LIN {X 0,Y 79.279,Z 952.165,A -85,B 0,C 180,E1 -27804.907,E2 -27804.907} C_VEL
LIN {X 0,Y 79.771,Z 953.591,A -85,B 0,C 180,E1 -27809.992,E2 -27809.992} C_VEL
LIN {X 0,Y 79.062,Z 954.279,A -85,B 0,C 180,E1 -27815.092,E2 -27815.092} C_VEL
LIN {X 0,Y 78.713,Z 954.565,A -85,B 0,C 180,E1 -27820.843,E2 -27820.843} C_VEL
LIN {X 0,Y 79.833,Z 953.994,A -85,B 0,C 180,E1 -27830.61,E2 -27830.61} C_VEL
LIN {X 0,Y 83.593,Z 951.93,A -85,B 0,C 180,E1 -27840.286,E2 -27840.286} C_VEL
LIN {X 0,Y 89.84,Z 948.411,A -85,B 0,C 180,E1 -27848.734,E2 -27848.734} C_VEL
LIN {X 0,Y 95.728,Z 944.699,A -85,B 0,C 180,E1 -27854.214,E2 -27854.214} C_VEL
LIN {X 0,Y 102.501,Z 939.995,A -85,B 0,C 180,E1 -27858.948,E2 -27858.948} C_VEL
LIN {X 0,Y 111.32,Z 933.115,A -85,B 0,C 180,E1 -27863.595,E2 -27863.595} C_VEL
LIN {X 0,Y 119.532,Z 925.735,A -85,B 0,C 180,E1 -27866.903,E2 -27866.903} C_VEL
LIN {X 0,Y 128.167,Z 916.709,A -85,B 0,C 180,E1 -27869.718,E2 -27869.718} C_VEL
LIN {X 0,Y 136.383,Z 906.598,A -85,B 0,C 180,E1 -27871.932,E2 -27871.932} C_VEL
LIN {X 0,Y 144.035,Z 895.124,A -85,B 0,C 180,E1 -27873.702,E2 -27873.702} C_VEL
LIN {X 0,Y 150.323,Z 883.666,A -85,B 0,C 180,E1 -27874.926,E2 -27874.926} C_VEL
LIN {X 0,Y 151.627,Z 880.908,A -85,B 0,C 180,E1 -27875.173,E2 -27875.173} C_VEL
LIN {X 0,Y 153.739,Z 875.695,A -85,B 0,C 180,E1 -27875.804,E2 -27875.804} C_VEL
LIN {X 0,Y 156.331,Z 867.052,A -85,B 0,C 180,E1 -27877.327,E2 -27877.327} C_VEL
LIN {X 0,Y 157.97,Z 860.05,A -85,B 0,C 180,E1 -27878.573,E2 -27878.573} C_VEL
LIN {X 0,Y 159.532,Z 852.692,A -85,B 0,C 180,E1 -27879.471,E2 -27879.471} C_VEL
LIN {X 0,Y 161.008,Z 844.469,A -85,B 0,C 180,E1 -27880.228,E2 -27880.228} C_VEL
LIN {X 0,Y 160.722,Z 839.975,A -85,B 0,C 180,E1 -27882.77,E2 -27882.77} C_VEL
LIN {X 0,Y 160.581,Z 836.729,A -85,B 0,C 180,E1 -27885.204,E2 -27885.204} C_VEL
LIN {X 0,Y 160.635,Z 833.991,A -85,B 0,C 180,E1 -27888.646,E2 -27888.646} C_VEL
LIN {X 0,Y 160.818,Z 833.978,A -85,B 0,C 180,E1 -27891.202,E2 -27891.202} C_VEL
LIN {X 0,Y 161.155,Z 834.602,A -85,B 0,C 180,E1 -27893.427,E2 -27893.427} C_VEL
LIN {X 0,Y 161.892,Z 837.639,A -85,B 0,C 180,E1 -27896.994,E2 -27896.994} C_VEL
LIN {X 0,Y 162.092,Z 838.711,A -85,B 0,C 180,E1 -27897.881,E2 -27897.881} C_VEL
LIN {X 0,Y 159.281,Z 851.041,A -85,B 0,C 180,E1 -27898.773,E2 -27898.773} C_VEL
LIN {X 0,Y 155.365,Z 862.808,A -85,B 0,C 180,E1 -27899.876,E2 -27899.876} C_VEL
LIN {X 0,Y 150.248,Z 874.331,A -85,B 0,C 180,E1 -27901.254,E2 -27901.254} C_VEL
LIN {X 0,Y 144.759,Z 884.196,A -85,B 0,C 180,E1 -27902.783,E2 -27902.783} C_VEL
LIN {X 0,Y 138.369,Z 893.655,A -85,B 0,C 180,E1 -27904.651,E2 -27904.651} C_VEL
LIN {X 0,Y 130.998,Z 902.698,A -85,B 0,C 180,E1 -27907.055,E2 -27907.055} C_VEL
LIN {X 0,Y 123.304,Z 910.519,A -85,B 0,C 180,E1 -27909.846,E2 -27909.846} C_VEL
LIN {X 0,Y 115.47,Z 917.219,A -85,B 0,C 180,E1 -27913.161,E2 -27913.161} C_VEL
LIN {X 0,Y 106.835,Z 923.354,A -85,B 0,C 180,E1 -27917.492,E2 -27917.492} C_VEL
LIN {X 0,Y 98.895,Z 927.947,A -85,B 0,C 180,E1 -27922.521,E2 -27922.521} C_VEL
LIN {X 0,Y 93.262,Z 930.598,A -85,B 0,C 180,E1 -27926.882,E2 -27926.882} C_VEL
LIN {X 0,Y 89.565,Z 932.059,A -85,B 0,C 180,E1 -27930.342,E2 -27930.342} C_VEL
LIN {X 0,Y 85.145,Z 933.404,A -85,B 0,C 180,E1 -27935.297,E2 -27935.297} C_VEL
LIN {X 0,Y 82.076,Z 934.072,A -85,B 0,C 180,E1 -27939.599,E2 -27939.599} C_VEL
LIN {X 0,Y 78.709,Z 934.361,A -85,B 0,C 180,E1 -27945.59,E2 -27945.59} C_VEL
LIN {X 0,Y 75.184,Z 933.555,A -85,B 0,C 180,E1 -27955.894,E2 -27955.894} C_VEL
LIN {X 0,Y 74.206,Z 932.448,A -85,B 0,C 180,E1 -27961.745,E2 -27961.745} C_VEL
LIN {X 0,Y 74.164,Z 929.647,A -85,B 0,C 180,E1 -27971.378,E2 -27971.378} C_VEL
LIN {X 0,Y 75.515,Z 926.299,A -85,B 0,C 180,E1 -27979.281,E2 -27979.281} C_VEL
LIN {X 0,Y 78.499,Z 921.25,A -85,B 0,C 180,E1 -27987.807,E2 -27987.807} C_VEL
LIN {X 0,Y 82.346,Z 915.432,A -85,B 0,C 180,E1 -27994.903,E2 -27994.903} C_VEL
LIN {X 0,Y 87.326,Z 907.86,A -85,B 0,C 180,E1 -28001.614,E2 -28001.614} C_VEL
LIN {X 0,Y 93.128,Z 898.429,A -85,B 0,C 180,E1 -28007.576,E2 -28007.576} C_VEL
LIN {X 0,Y 98.653,Z 888.378,A -85,B 0,C 180,E1 -28012.16,E2 -28012.16} C_VEL
LIN {X 0,Y 103.614,Z 877.982,A -85,B 0,C 180,E1 -28015.627,E2 -28015.627} C_VEL
LIN {X 0,Y 108.336,Z 866.102,A -85,B 0,C 180,E1 -28018.589,E2 -28018.589} C_VEL
LIN {X 0,Y 111.893,Z 854.99,A -85,B 0,C 180,E1 -28020.613,E2 -28020.613} C_VEL
LIN {X 0,Y 114.994,Z 841.627,A -85,B 0,C 180,E1 -28022.418,E2 -28022.418} C_VEL
LIN {X 0,Y 116.954,Z 828.557,A -85,B 0,C 180,E1 -28023.645,E2 -28023.645} C_VEL
LIN {X 0,Y 117.953,Z 816.094,A -85,B 0,C 180,E1 -28024.436,E2 -28024.436} C_VEL
LIN {X 0,Y 114.276,Z 825.052,A -85,B 0,C 180,E1 -28025.793,E2 -28025.793} C_VEL
LIN {X 0,Y 110.929,Z 830.932,A -85,B 0,C 180,E1 -28027.258,E2 -28027.258} C_VEL
LIN {X 0,Y 109.143,Z 833.439,A -85,B 0,C 180,E1 -28028.112,E2 -28028.112} C_VEL
LIN {X 0,Y 104.574,Z 843.452,A -85,B 0,C 180,E1 -28029.387,E2 -28029.387} C_VEL
LIN {X 0,Y 100.024,Z 850.982,A -85,B 0,C 180,E1 -28030.944,E2 -28030.944} C_VEL
LIN {X 0,Y 95.912,Z 856.125,A -85,B 0,C 180,E1 -28032.881,E2 -28032.881} C_VEL
LIN {X 0,Y 93.49,Z 858.415,A -85,B 0,C 180,E1 -28034.425,E2 -28034.425} C_VEL
LIN {X 0,Y 91.256,Z 860.296,A -85,B 0,C 180,E1 -28036.12,E2 -28036.12} C_VEL
LIN {X 0,Y 87.235,Z 865.271,A -85,B 0,C 180,E1 -28038.343,E2 -28038.343} C_VEL
LIN {X 0,Y 83.714,Z 868.947,A -85,B 0,C 180,E1 -28040.975,E2 -28040.975} C_VEL
LIN {X 0,Y 80.182,Z 871.594,A -85,B 0,C 180,E1 -28045.267,E2 -28045.267} C_VEL
LIN {X 0,Y 77.18,Z 875.194,A -85,B 0,C 180,E1 -28048.004,E2 -28048.004} C_VEL
LIN {X 0,Y 75.913,Z 876.588,A -85,B 0,C 180,E1 -28049.529,E2 -28049.529} C_VEL
LIN {X 0,Y 74.562,Z 877.879,A -85,B 0,C 180,E1 -28051.881,E2 -28051.881} C_VEL
LIN {X 0,Y 73.899,Z 878.573,A -85,B 0,C 180,E1 -28054.661,E2 -28054.661} C_VEL
LIN {X 0,Y 73.738,Z 880.411,A -85,B 0,C 180,E1 -28056.476,E2 -28056.476} C_VEL
LIN {X 0,Y 73.167,Z 894.524,A -85,B 0,C 180,E1 -28066.167,E2 -28066.167} C_VEL
LIN {X 0,Y 74.081,Z 904.378,A -85,B 0,C 180,E1 -28074.555,E2 -28074.555} C_VEL
LIN {X 0,Y 75.997,Z 911.495,A -85,B 0,C 180,E1 -28081.324,E2 -28081.324} C_VEL
LIN {X 0,Y 79.638,Z 918.739,A -85,B 0,C 180,E1 -28088.883,E2 -28088.883} C_VEL
LIN {X 0,Y 83.592,Z 923.927,A -85,B 0,C 180,E1 -28094.608,E2 -28094.608} C_VEL
LIN {X 0,Y 90.963,Z 930.199,A -85,B 0,C 180,E1 -28101.99,E2 -28101.99} C_VEL
LIN {X 0,Y 98.835,Z 934.682,A -85,B 0,C 180,E1 -28107.529,E2 -28107.529} C_VEL
LIN {X 0,Y 106.808,Z 937.884,A -85,B 0,C 180,E1 -28111.762,E2 -28111.762} C_VEL
LIN {X 0,Y 108.246,Z 938.311,A -85,B 0,C 180,E1 -28112.421,E2 -28112.421} C_VEL
LIN {X 0,Y 109.349,Z 938.789,A -85,B 0,C 180,E1 -28113.32,E2 -28113.32} C_VEL
LIN {X 0,Y 103.989,Z 938.934,A -85,B 0,C 180,E1 -28115.796,E2 -28115.796} C_VEL
LIN {X 0,Y 92.354,Z 938.024,A -85,B 0,C 180,E1 -28123.226,E2 -28123.226} C_VEL
LIN {X 0,Y 86.202,Z 936.736,A -85,B 0,C 180,E1 -28129.281,E2 -28129.281} C_VEL
LIN {X 0,Y 81.237,Z 934.962,A -85,B 0,C 180,E1 -28136.706,E2 -28136.706} C_VEL
LIN {X 0,Y 75.515,Z 941.92,A -85,B 0,C 180,E1 -28145.233,E2 -28145.233} C_VEL
LIN {X 0,Y 72.937,Z 946.473,A -85,B 0,C 180,E1 -28153.189,E2 -28153.189} C_VEL
LIN {X 0,Y 72.199,Z 948.887,A -85,B 0,C 180,E1 -28158.765,E2 -28158.765} C_VEL
LIN {X 0,Y 72.228,Z 950.867,A -85,B 0,C 180,E1 -28164.408,E2 -28164.408} C_VEL
LIN {X 0,Y 72.701,Z 952.378,A -85,B 0,C 180,E1 -28169.992,E2 -28169.992} C_VEL
LIN {X 0,Y 71.986,Z 953.129,A -85,B 0,C 180,E1 -28175.594,E2 -28175.594} C_VEL
LIN {X 0,Y 72.059,Z 953.393,A -85,B 0,C 180,E1 -28187.004,E2 -28187.004} C_VEL
LIN {X 0,Y 74.972,Z 952.22,A -85,B 0,C 180,E1 -28197.941,E2 -28197.941} C_VEL
LIN {X 0,Y 80.664,Z 949.567,A -85,B 0,C 180,E1 -28207.572,E2 -28207.572} C_VEL
LIN {X 0,Y 88.532,Z 945.403,A -85,B 0,C 180,E1 -28215.588,E2 -28215.588} C_VEL
LIN {X 0,Y 95.468,Z 941.154,A -85,B 0,C 180,E1 -28220.611,E2 -28220.611} C_VEL
LIN {X 0,Y 104.515,Z 934.899,A -85,B 0,C 180,E1 -28225.45,E2 -28225.45} C_VEL
LIN {X 0,Y 112.899,Z 928.191,A -85,B 0,C 180,E1 -28228.853,E2 -28228.853} C_VEL
LIN {X 0,Y 121.712,Z 919.984,A -85,B 0,C 180,E1 -28231.701,E2 -28231.701} C_VEL
LIN {X 0,Y 129.317,Z 911.73,A -85,B 0,C 180,E1 -28233.72,E2 -28233.72} C_VEL
LIN {X 0,Y 137.109,Z 901.774,A -85,B 0,C 180,E1 -28235.472,E2 -28235.472} C_VEL
LIN {X 0,Y 144.256,Z 890.754,A -85,B 0,C 180,E1 -28236.851,E2 -28236.851} C_VEL
LIN {X 0,Y 150.705,Z 878.352,A -85,B 0,C 180,E1 -28237.938,E2 -28237.938} C_VEL
LIN {X 0,Y 155.89,Z 865.509,A -85,B 0,C 180,E1 -28238.754,E2 -28238.754} C_VEL
LIN {X 0,Y 159.26,Z 854.005,A -85,B 0,C 180,E1 -28239.36,E2 -28239.36} C_VEL
LIN {X 0,Y 159.532,Z 852.692,A -85,B 0,C 180,E1 -28239.471,E2 -28239.471} C_VEL
LIN {X 0,Y 159.946,Z 849.938,A -85,B 0,C 180,E1 -28239.994,E2 -28239.994} C_VEL
LIN {X 0,Y 160.004,Z 847.475,A -85,B 0,C 180,E1 -28241.079,E2 -28241.079} C_VEL
LIN {X 0,Y 159.847,Z 846.084,A -85,B 0,C 180,E1 -28242.162,E2 -28242.162} C_VEL
LIN {X 0,Y 159.275,Z 843.099,A -85,B 0,C 180,E1 -28246.31,E2 -28246.31} C_VEL
LIN {X 0,Y 159.466,Z 840.92,A -85,B 0,C 180,E1 -28249.205,E2 -28249.205} C_VEL
LIN {X 0,Y 159.772,Z 841.293,A -85,B 0,C 180,E1 -28252.735,E2 -28252.735} C_VEL
LIN {X 0,Y 160.047,Z 843.578,A -85,B 0,C 180,E1 -28255.673,E2 -28255.673} C_VEL
LIN {X 0,Y 156.564,Z 856.366,A -85,B 0,C 180,E1 -28256.632,E2 -28256.632} C_VEL
LIN {X 0,Y 152.122,Z 868.038,A -85,B 0,C 180,E1 -28257.762,E2 -28257.762} C_VEL
LIN {X 0,Y 146.181,Z 879.81,A -85,B 0,C 180,E1 -28259.239,E2 -28259.239} C_VEL
LIN {X 0,Y 139.688,Z 890.07,A -85,B 0,C 180,E1 -28260.93,E2 -28260.93} C_VEL
LIN {X 0,Y 132.124,Z 899.819,A -85,B 0,C 180,E1 -28263.05,E2 -28263.05} C_VEL
LIN {X 0,Y 123.593,Z 908.767,A -85,B 0,C 180,E1 -28265.733,E2 -28265.733} C_VEL
LIN {X 0,Y 115.513,Z 915.842,A -85,B 0,C 180,E1 -28268.669,E2 -28268.669} C_VEL
LIN {X 0,Y 107.741,Z 921.534,A -85,B 0,C 180,E1 -28271.944,E2 -28271.944} C_VEL
LIN {X 0,Y 98.976,Z 926.863,A -85,B 0,C 180,E1 -28276.501,E2 -28276.501} C_VEL
LIN {X 0,Y 90.82,Z 930.778,A -85,B 0,C 180,E1 -28281.8,E2 -28281.8} C_VEL
LIN {X 0,Y 85.87,Z 932.677,A -85,B 0,C 180,E1 -28285.821,E2 -28285.821} C_VEL
LIN {X 0,Y 79.956,Z 934.411,A -85,B 0,C 180,E1 -28291.831,E2 -28291.831} C_VEL
LIN {X 0,Y 73.875,Z 935.38,A -85,B 0,C 180,E1 -28300.454,E2 -28300.454} C_VEL
LIN {X 0,Y 71.034,Z 935.332,A -85,B 0,C 180,E1 -28306.178,E2 -28306.178} C_VEL
LIN {X 0,Y 68.091,Z 934.338,A -85,B 0,C 180,E1 -28315.663,E2 -28315.663} C_VEL
LIN {X 0,Y 66.919,Z 932.385,A -85,B 0,C 180,E1 -28325.17,E2 -28325.17} C_VEL
LIN {X 0,Y 67.522,Z 929.319,A -85,B 0,C 180,E1 -28334.927,E2 -28334.927} C_VEL
LIN {X 0,Y 69.752,Z 925.135,A -85,B 0,C 180,E1 -28344.226,E2 -28344.226} C_VEL
LIN {X 0,Y 73.409,Z 919.738,A -85,B 0,C 180,E1 -28352.752,E2 -28352.752} C_VEL
LIN {X 0,Y 78.223,Z 912.997,A -85,B 0,C 180,E1 -28360.359,E2 -28360.359} C_VEL
LIN {X 0,Y 84.029,Z 904.553,A -85,B 0,C 180,E1 -28367.029,E2 -28367.029} C_VEL
LIN {X 0,Y 89.447,Z 895.965,A -85,B 0,C 180,E1 -28371.921,E2 -28371.921} C_VEL
LIN {X 0,Y 95.312,Z 885.491,A -85,B 0,C 180,E1 -28376.265,E2 -28376.265} C_VEL
LIN {X 0,Y 100.146,Z 875.166,A -85,B 0,C 180,E1 -28379.429,E2 -28379.429} C_VEL
LIN {X 0,Y 104.549,Z 863.95,A -85,B 0,C 180,E1 -28381.97,E2 -28381.97} C_VEL
LIN {X 0,Y 108.442,Z 851.317,A -85,B 0,C 180,E1 -28384.077,E2 -28384.077} C_VEL
LIN {X 0,Y 110.945,Z 840.041,A -85,B 0,C 180,E1 -28385.451,E2 -28385.451} C_VEL
LIN {X 0,Y 110.858,Z 839.871,A -85,B 0,C 180,E1 -28385.548,E2 -28385.548} C_VEL
LIN {X 0,Y 106.257,Z 848.445,A -85,B 0,C 180,E1 -28386.539,E2 -28386.539} C_VEL
LIN {X 0,Y 100.979,Z 856.035,A -85,B 0,C 180,E1 -28388.061,E2 -28388.061} C_VEL
LIN {X 0,Y 96.988,Z 860.539,A -85,B 0,C 180,E1 -28389.653,E2 -28389.653} C_VEL
LIN {X 0,Y 93.696,Z 863.529,A -85,B 0,C 180,E1 -28391.401,E2 -28391.401} C_VEL
LIN {X 0,Y 91.228,Z 865.472,A -85,B 0,C 180,E1 -28392.956,E2 -28392.956} C_VEL
LIN {X 0,Y 86.27,Z 870.854,A -85,B 0,C 180,E1 -28395.359,E2 -28395.359} C_VEL
LIN {X 0,Y 83.098,Z 873.771,A -85,B 0,C 180,E1 -28397.42,E2 -28397.42} C_VEL
LIN {X 0,Y 78.992,Z 876.735,A -85,B 0,C 180,E1 -28401.478,E2 -28401.478} C_VEL
LIN {X 0,Y 74.441,Z 881.158,A -85,B 0,C 180,E1 -28405.495,E2 -28405.495} C_VEL
LIN {X 0,Y 72.659,Z 882.721,A -85,B 0,C 180,E1 -28407.858,E2 -28407.858} C_VEL
LIN {X 0,Y 69.991,Z 884.836,A -85,B 0,C 180,E1 -28413.136,E2 -28413.136} C_VEL
LIN {X 0,Y 68.251,Z 886.856,A -85,B 0,C 180,E1 -28415.675,E2 -28415.675} C_VEL
LIN {X 0,Y 66.971,Z 888.374,A -85,B 0,C 180,E1 -28418.45,E2 -28418.45} C_VEL
LIN {X 0,Y 66.147,Z 889.514,A -85,B 0,C 180,E1 -28422.267,E2 -28422.267} C_VEL
LIN {X 0,Y 66.234,Z 890.424,A -85,B 0,C 180,E1 -28424.728,E2 -28424.728} C_VEL
LIN {X 0,Y 66.388,Z 893.57,A -85,B 0,C 180,E1 -28427.775,E2 -28427.775} C_VEL
LIN {X 0,Y 67.982,Z 905.362,A -85,B 0,C 180,E1 -28438.518,E2 -28438.518} C_VEL
LIN {X 0,Y 70.688,Z 912.767,A -85,B 0,C 180,E1 -28446.087,E2 -28446.087} C_VEL
LIN {X 0,Y 75.721,Z 920.736,A -85,B 0,C 180,E1 -28454.787,E2 -28454.787} C_VEL
LIN {X 0,Y 80.472,Z 925.78,A -85,B 0,C 180,E1 -28460.446,E2 -28460.446} C_VEL
LIN {X 0,Y 87.334,Z 930.984,A -85,B 0,C 180,E1 -28466.311,E2 -28466.311} C_VEL
LIN {X 0,Y 97.218,Z 936.155,A -85,B 0,C 180,E1 -28472.367,E2 -28472.367} C_VEL
LIN {X 0,Y 98.251,Z 936.566,A -85,B 0,C 180,E1 -28472.863,E2 -28472.863} C_VEL
LIN {X 0,Y 96.613,Z 936.715,A -85,B 0,C 180,E1 -28474.401,E2 -28474.401} C_VEL
LIN {X 0,Y 85.32,Z 935.166,A -85,B 0,C 180,E1 -28482.144,E2 -28482.144} C_VEL
LIN {X 0,Y 76.325,Z 932.435,A -85,B 0,C 180,E1 -28493.02,E2 -28493.02} C_VEL
LIN {X 0,Y 70.691,Z 938.584,A -85,B 0,C 180,E1 -28500.183,E2 -28500.183} C_VEL
LIN {X 0,Y 66.972,Z 943.591,A -85,B 0,C 180,E1 -28508.442,E2 -28508.442} C_VEL
LIN {X 0,Y 65.243,Z 947.53,A -85,B 0,C 180,E1 -28517.549,E2 -28517.549} C_VEL
LIN {X 0,Y 65.161,Z 949.564,A -85,B 0,C 180,E1 -28523.799,E2 -28523.799} C_VEL
LIN {X 0,Y 65.632,Z 951.133,A -85,B 0,C 180,E1 -28529.991,E2 -28529.991} C_VEL
LIN {X 0,Y 64.911,Z 951.962,A -85,B 0,C 180,E1 -28536.206,E2 -28536.206} C_VEL
LIN {X 0,Y 64.715,Z 952.342,A -85,B 0,C 180,E1 -28542.535,E2 -28542.535} C_VEL
LIN {X 0,Y 66.626,Z 951.981,A -85,B 0,C 180,E1 -28554.947,E2 -28554.947} C_VEL
LIN {X 0,Y 71.626,Z 950.218,A -85,B 0,C 180,E1 -28566.056,E2 -28566.056} C_VEL
LIN {X 0,Y 77.374,Z 947.796,A -85,B 0,C 180,E1 -28573.395,E2 -28573.395} C_VEL
LIN {X 0,Y 86.06,Z 943.489,A -85,B 0,C 180,E1 -28580.867,E2 -28580.867} C_VEL
LIN {X 0,Y 93.751,Z 939.063,A -85,B 0,C 180,E1 -28585.537,E2 -28585.537} C_VEL
LIN {X 0,Y 103.523,Z 932.504,A -85,B 0,C 180,E1 -28589.936,E2 -28589.936} C_VEL
LIN {X 0,Y 112.417,Z 925.523,A -85,B 0,C 180,E1 -28592.971,E2 -28592.971} C_VEL
LIN {X 0,Y 121.626,Z 917.004,A -85,B 0,C 180,E1 -28595.505,E2 -28595.505} C_VEL
LIN {X 0,Y 129.525,Z 908.398,A -85,B 0,C 180,E1 -28597.269,E2 -28597.269} C_VEL
LIN {X 0,Y 137.552,Z 897.919,A -85,B 0,C 180,E1 -28598.807,E2 -28598.807} C_VEL
LIN {X 0,Y 144.912,Z 886.252,A -85,B 0,C 180,E1 -28599.981,E2 -28599.981} C_VEL
LIN {X 0,Y 150.561,Z 875.083,A -85,B 0,C 180,E1 -28600.797,E2 -28600.797} C_VEL
LIN {X 0,Y 155.629,Z 861.973,A -85,B 0,C 180,E1 -28601.488,E2 -28601.488} C_VEL
LIN {X 0,Y 157.767,Z 854.772,A -85,B 0,C 180,E1 -28601.854,E2 -28601.854} C_VEL
LIN {X 0,Y 159.163,Z 848.548,A -85,B 0,C 180,E1 -28602.411,E2 -28602.411} C_VEL
LIN {X 0,Y 159.186,Z 845.306,A -85,B 0,C 180,E1 -28604.518,E2 -28604.518} C_VEL
LIN {X 0,Y 159.275,Z 843.099,A -85,B 0,C 180,E1 -28606.31,E2 -28606.31} C_VEL
LIN {X 0,Y 159.124,Z 843.309,A -85,B 0,C 180,E1 -28607.171,E2 -28607.171} C_VEL
LIN {X 0,Y 158.676,Z 845.012,A -85,B 0,C 180,E1 -28608.178,E2 -28608.178} C_VEL
LIN {X 0,Y 158.009,Z 847.51,A -85,B 0,C 180,E1 -28609.565,E2 -28609.565} C_VEL
LIN {X 0,Y 157.945,Z 847.809,A -85,B 0,C 180,E1 -28610.096,E2 -28610.096} C_VEL
LIN {X 0,Y 158.073,Z 848.342,A -85,B 0,C 180,E1 -28612.57,E2 -28612.57} C_VEL
LIN {X 0,Y 158.048,Z 848.996,A -85,B 0,C 180,E1 -28613.449,E2 -28613.449} C_VEL
LIN {X 0,Y 154.112,Z 861.259,A -85,B 0,C 180,E1 -28614.403,E2 -28614.403} C_VEL
LIN {X 0,Y 149.137,Z 872.75,A -85,B 0,C 180,E1 -28615.532,E2 -28615.532} C_VEL
LIN {X 0,Y 143.167,Z 883.56,A -85,B 0,C 180,E1 -28616.895,E2 -28616.895} C_VEL
LIN {X 0,Y 136.2,Z 893.642,A -85,B 0,C 180,E1 -28618.548,E2 -28618.548} C_VEL
LIN {X 0,Y 127.588,Z 903.776,A -85,B 0,C 180,E1 -28620.804,E2 -28620.804} C_VEL
LIN {X 0,Y 118.811,Z 912.164,A -85,B 0,C 180,E1 -28623.392,E2 -28623.392} C_VEL
LIN {X 0,Y 109.643,Z 919.34,A -85,B 0,C 180,E1 -28626.587,E2 -28626.587} C_VEL
LIN {X 0,Y 100.071,Z 925.445,A -85,B 0,C 180,E1 -28630.546,E2 -28630.546} C_VEL
LIN {X 0,Y 91.074,Z 930.039,A -85,B 0,C 180,E1 -28635.318,E2 -28635.318} C_VEL
LIN {X 0,Y 82.761,Z 933.303,A -85,B 0,C 180,E1 -28640.936,E2 -28640.936} C_VEL
LIN {X 0,Y 75.086,Z 935.437,A -85,B 0,C 180,E1 -28647.905,E2 -28647.905} C_VEL
LIN {X 0,Y 66.97,Z 936.458,A -85,B 0,C 180,E1 -28659.026,E2 -28659.026} C_VEL
LIN {X 0,Y 62.979,Z 936.037,A -85,B 0,C 180,E1 -28667.98,E2 -28667.98} C_VEL
LIN {X 0,Y 61.101,Z 935.16,A -85,B 0,C 180,E1 -28674.905,E2 -28674.905} C_VEL
LIN {X 0,Y 60.064,Z 933.858,A -85,B 0,C 180,E1 -28682.105,E2 -28682.105} C_VEL
LIN {X 0,Y 60.192,Z 930.952,A -85,B 0,C 180,E1 -28693.181,E2 -28693.181} C_VEL
LIN {X 0,Y 62.199,Z 927.02,A -85,B 0,C 180,E1 -28703.522,E2 -28703.522} C_VEL
LIN {X 0,Y 66.656,Z 920.821,A -85,B 0,C 180,E1 -28714.545,E2 -28714.545} C_VEL
LIN {X 0,Y 72.157,Z 913.711,A -85,B 0,C 180,E1 -28723.091,E2 -28723.091} C_VEL
LIN {X 0,Y 78.081,Z 905.657,A -85,B 0,C 180,E1 -28729.735,E2 -28729.735} C_VEL
LIN {X 0,Y 84.742,Z 895.704,A -85,B 0,C 180,E1 -28735.471,E2 -28735.471} C_VEL
LIN {X 0,Y 90.705,Z 885.425,A -85,B 0,C 180,E1 -28739.608,E2 -28739.608} C_VEL
LIN {X 0,Y 95.855,Z 874.862,A -85,B 0,C 180,E1 -28742.74,E2 -28742.74} C_VEL
LIN {X 0,Y 99.977,Z 864.718,A -85,B 0,C 180,E1 -28744.989,E2 -28744.989} C_VEL
LIN {X 0,Y 99.533,Z 863.526,A -85,B 0,C 180,E1 -28745.944,E2 -28745.944} C_VEL
LIN {X 0,Y 95.336,Z 867.392,A -85,B 0,C 180,E1 -28747.581,E2 -28747.581} C_VEL
LIN {X 0,Y 91.316,Z 870.43,A -85,B 0,C 180,E1 -28749.678,E2 -28749.678} C_VEL
LIN {X 0,Y 86.778,Z 874.907,A -85,B 0,C 180,E1 -28751.483,E2 -28751.483} C_VEL
LIN {X 0,Y 82.629,Z 878.393,A -85,B 0,C 180,E1 -28753.699,E2 -28753.699} C_VEL
LIN {X 0,Y 77.991,Z 881.571,A -85,B 0,C 180,E1 -28757.479,E2 -28757.479} C_VEL
LIN {X 0,Y 73.08,Z 885.614,A -85,B 0,C 180,E1 -28761.309,E2 -28761.309} C_VEL
LIN {X 0,Y 69.144,Z 888.583,A -85,B 0,C 180,E1 -28766.009,E2 -28766.009} C_VEL
LIN {X 0,Y 67.602,Z 889.641,A -85,B 0,C 180,E1 -28768.679,E2 -28768.679} C_VEL
LIN {X 0,Y 64.192,Z 892.779,A -85,B 0,C 180,E1 -28774.026,E2 -28774.026} C_VEL
LIN {X 0,Y 62.928,Z 894.051,A -85,B 0,C 180,E1 -28776.989,E2 -28776.989} C_VEL
LIN {X 0,Y 61.292,Z 896.079,A -85,B 0,C 180,E1 -28783.756,E2 -28783.756} C_VEL
LIN {X 0,Y 60.372,Z 897.468,A -85,B 0,C 180,E1 -28786.536,E2 -28786.536} C_VEL
LIN {X 0,Y 59.79,Z 898.71,A -85,B 0,C 180,E1 -28789.843,E2 -28789.843} C_VEL
LIN {X 0,Y 59.749,Z 899.557,A -85,B 0,C 180,E1 -28793.244,E2 -28793.244} C_VEL
LIN {X 0,Y 60.375,Z 900.108,A -85,B 0,C 180,E1 -28796.245,E2 -28796.245} C_VEL
LIN {X 0,Y 60.934,Z 901.592,A -85,B 0,C 180,E1 -28798.347,E2 -28798.347} C_VEL
LIN {X 0,Y 65.275,Z 912.94,A -85,B 0,C 180,E1 -28810.442,E2 -28810.442} C_VEL
LIN {X 0,Y 71.679,Z 921.553,A -85,B 0,C 180,E1 -28820.069,E2 -28820.069} C_VEL
LIN {X 0,Y 78.318,Z 927.587,A -85,B 0,C 180,E1 -28826.658,E2 -28826.658} C_VEL
LIN {X 0,Y 87.399,Z 933.373,A -85,B 0,C 180,E1 -28832.873,E2 -28832.873} C_VEL
LIN {X 0,Y 86.265,Z 933.593,A -85,B 0,C 180,E1 -28834.77,E2 -28834.77} C_VEL
LIN {X 0,Y 76.676,Z 931.326,A -85,B 0,C 180,E1 -28842.828,E2 -28842.828} C_VEL
LIN {X 0,Y 71.992,Z 929.747,A -85,B 0,C 180,E1 -28848.77,E2 -28848.77} C_VEL
LIN {X 0,Y 64.713,Z 936.949,A -85,B 0,C 180,E1 -28857.1,E2 -28857.1} C_VEL
LIN {X 0,Y 60.471,Z 942.086,A -85,B 0,C 180,E1 -28865.987,E2 -28865.987} C_VEL
LIN {X 0,Y 58.336,Z 946.136,A -85,B 0,C 180,E1 -28876.047,E2 -28876.047} C_VEL
LIN {X 0,Y 58.108,Z 948.251,A -85,B 0,C 180,E1 -28883.043,E2 -28883.043} C_VEL
LIN {X 0,Y 58.559,Z 949.877,A -85,B 0,C 180,E1 -28889.99,E2 -28889.99} C_VEL
LIN {X 0,Y 57.849,Z 950.749,A -85,B 0,C 180,E1 -28896.968,E2 -28896.968} C_VEL
LIN {X 0,Y 58.553,Z 951.281,A -85,B 0,C 180,E1 -28911.094,E2 -28911.094} C_VEL
LIN {X 0,Y 62.686,Z 950.317,A -85,B 0,C 180,E1 -28924.083,E2 -28924.083} C_VEL
LIN {X 0,Y 69.893,Z 947.977,A -85,B 0,C 180,E1 -28934.726,E2 -28934.726} C_VEL
LIN {X 0,Y 76.724,Z 945.216,A -85,B 0,C 180,E1 -28941.12,E2 -28941.12} C_VEL
LIN {X 0,Y 84.39,Z 941.549,A -85,B 0,C 180,E1 -28946.374,E2 -28946.374} C_VEL
LIN {X 0,Y 92.763,Z 936.904,A -85,B 0,C 180,E1 -28950.593,E2 -28950.593} C_VEL
LIN {X 0,Y 103.17,Z 930.115,A -85,B 0,C 180,E1 -28954.487,E2 -28954.487} C_VEL
LIN {X 0,Y 112.499,Z 922.874,A -85,B 0,C 180,E1 -28957.126,E2 -28957.126} C_VEL
LIN {X 0,Y 122.077,Z 913.974,A -85,B 0,C 180,E1 -28959.297,E2 -28959.297} C_VEL
LIN {X 0,Y 130.249,Z 904.973,A -85,B 0,C 180,E1 -28960.766,E2 -28960.766} C_VEL
LIN {X 0,Y 137.655,Z 895.204,A -85,B 0,C 180,E1 -28961.956,E2 -28961.956} C_VEL
LIN {X 0,Y 144.32,Z 884.619,A -85,B 0,C 180,E1 -28962.863,E2 -28962.863} C_VEL
LIN {X 0,Y 150.607,Z 872.033,A -85,B 0,C 180,E1 -28963.613,E2 -28963.613} C_VEL
LIN {X 0,Y 155.392,Z 859.467,A -85,B 0,C 180,E1 -28964.171,E2 -28964.171} C_VEL
LIN {X 0,Y 157.182,Z 853.329,A -85,B 0,C 180,E1 -28964.577,E2 -28964.577} C_VEL
LIN {X 0,Y 157.344,Z 852.643,A -85,B 0,C 180,E1 -28964.731,E2 -28964.731} C_VEL
LIN {X 0,Y 157.651,Z 849.644,A -85,B 0,C 180,E1 -28967.121,E2 -28967.121} C_VEL
LIN {X 0,Y 157.921,Z 847.823,A -85,B 0,C 180,E1 -28969.43,E2 -28969.43} C_VEL
LIN {X 0,Y 157.945,Z 847.809,A -85,B 0,C 180,E1 -28970.096,E2 -28970.096} C_VEL
LIN {X 0,Y 157.78,Z 848.668,A -85,B 0,C 180,E1 -28970.865,E2 -28970.865} C_VEL
LIN {X 0,Y 157.337,Z 850.447,A -85,B 0,C 180,E1 -28971.428,E2 -28971.428} C_VEL
LIN {X 0,Y 156.342,Z 853.974,A -85,B 0,C 180,E1 -28971.93,E2 -28971.93} C_VEL
LIN {X 0,Y 153.793,Z 861.299,A -85,B 0,C 180,E1 -28972.05,E2 -28972.05} C_VEL
LIN {X 0,Y 151.357,Z 867.22,A -85,B 0,C 180,E1 -28972.241,E2 -28972.241} C_VEL
LIN {X 0,Y 145.933,Z 878.177,A -85,B 0,C 180,E1 -28973.314,E2 -28973.314} C_VEL
LIN {X 0,Y 139.393,Z 888.685,A -85,B 0,C 180,E1 -28974.673,E2 -28974.673} C_VEL
LIN {X 0,Y 132.44,Z 897.774,A -85,B 0,C 180,E1 -28976.18,E2 -28976.18} C_VEL
LIN {X 0,Y 124.812,Z 906.04,A -85,B 0,C 180,E1 -28978,E2 -28978} C_VEL
LIN {X 0,Y 117.197,Z 913.003,A -85,B 0,C 180,E1 -28980.001,E2 -28980.001} C_VEL
LIN {X 0,Y 107.318,Z 920.446,A -85,B 0,C 180,E1 -28983.057,E2 -28983.057} C_VEL
LIN {X 0,Y 98.938,Z 925.62,A -85,B 0,C 180,E1 -28986.085,E2 -28986.085} C_VEL
LIN {X 0,Y 89.327,Z 930.431,A -85,B 0,C 180,E1 -28990.473,E2 -28990.473} C_VEL
LIN {X 0,Y 80.293,Z 933.916,A -85,B 0,C 180,E1 -28995.701,E2 -28995.701} C_VEL
LIN {X 0,Y 70.61,Z 936.464,A -85,B 0,C 180,E1 -29003.463,E2 -29003.463} C_VEL
LIN {X 0,Y 64.873,Z 937.337,A -85,B 0,C 180,E1 -29009.945,E2 -29009.945} C_VEL
LIN {X 0,Y 60.801,Z 937.5,A -85,B 0,C 180,E1 -29016.007,E2 -29016.007} C_VEL
LIN {X 0,Y 57.455,Z 937.228,A -85,B 0,C 180,E1 -29022.799,E2 -29022.799} C_VEL
LIN {X 0,Y 54.953,Z 936.484,A -85,B 0,C 180,E1 -29030.263,E2 -29030.263} C_VEL
LIN {X 0,Y 53.407,Z 935.26,A -85,B 0,C 180,E1 -29038.253,E2 -29038.253} C_VEL
LIN {X 0,Y 52.826,Z 933.089,A -85,B 0,C 180,E1 -29048.64,E2 -29048.64} C_VEL
LIN {X 0,Y 54.663,Z 928.805,A -85,B 0,C 180,E1 -29062.624,E2 -29062.624} C_VEL
LIN {X 0,Y 58.381,Z 923.852,A -85,B 0,C 180,E1 -29073.461,E2 -29073.461} C_VEL
LIN {X 0,Y 63.636,Z 917.583,A -85,B 0,C 180,E1 -29082.77,E2 -29082.77} C_VEL
LIN {X 0,Y 70.016,Z 909.754,A -85,B 0,C 180,E1 -29090.577,E2 -29090.577} C_VEL
LIN {X 0,Y 76.001,Z 901.813,A -85,B 0,C 180,E1 -29096.064,E2 -29096.064} C_VEL
LIN {X 0,Y 82.398,Z 892.238,A -85,B 0,C 180,E1 -29100.789,E2 -29100.789} C_VEL
LIN {X 0,Y 88.446,Z 881.646,A -85,B 0,C 180,E1 -29104.445,E2 -29104.445} C_VEL
LIN {X 0,Y 90.628,Z 877.258,A -85,B 0,C 180,E1 -29105.682,E2 -29105.682} C_VEL
LIN {X 0,Y 90.904,Z 875.765,A -85,B 0,C 180,E1 -29106.464,E2 -29106.464} C_VEL
LIN {X 0,Y 85.297,Z 880.588,A -85,B 0,C 180,E1 -29108.486,E2 -29108.486} C_VEL
LIN {X 0,Y 82.361,Z 882.829,A -85,B 0,C 180,E1 -29109.825,E2 -29109.825} C_VEL
LIN {X 0,Y 74.655,Z 887.82,A -85,B 0,C 180,E1 -29115.084,E2 -29115.084} C_VEL
LIN {X 0,Y 69.558,Z 891.536,A -85,B 0,C 180,E1 -29118.946,E2 -29118.946} C_VEL
LIN {X 0,Y 63.599,Z 895.417,A -85,B 0,C 180,E1 -29126.458,E2 -29126.458} C_VEL
LIN {X 0,Y 59.988,Z 898.327,A -85,B 0,C 180,E1 -29132.053,E2 -29132.053} C_VEL
LIN {X 0,Y 56.658,Z 901.513,A -85,B 0,C 180,E1 -29141.933,E2 -29141.933} C_VEL
LIN {X 0,Y 55.644,Z 902.857,A -85,B 0,C 180,E1 -29145.367,E2 -29145.367} C_VEL
LIN {X 0,Y 56.216,Z 908.518,A -85,B 0,C 180,E1 -29167.181,E2 -29167.181} C_VEL
LIN {X 0,Y 57.972,Z 909.359,A -85,B 0,C 180,E1 -29171.084,E2 -29171.084} C_VEL
LIN {X 0,Y 68.287,Z 922.317,A -85,B 0,C 180,E1 -29185.938,E2 -29185.938} C_VEL
LIN {X 0,Y 77.15,Z 929.264,A -85,B 0,C 180,E1 -29193.131,E2 -29193.131} C_VEL
LIN {X 0,Y 77.909,Z 929.754,A -85,B 0,C 180,E1 -29193.633,E2 -29193.633} C_VEL
LIN {X 0,Y 77.081,Z 929.736,A -85,B 0,C 180,E1 -29194.843,E2 -29194.843} C_VEL
LIN {X 0,Y 67.951,Z 926.989,A -85,B 0,C 180,E1 -29204.137,E2 -29204.137} C_VEL
LIN {X 0,Y 59.966,Z 934.294,A -85,B 0,C 180,E1 -29212.014,E2 -29212.014} C_VEL
LIN {X 0,Y 54.115,Z 940.529,A -85,B 0,C 180,E1 -29222.952,E2 -29222.952} C_VEL
LIN {X 0,Y 51.508,Z 944.7,A -85,B 0,C 180,E1 -29234.152,E2 -29234.152} C_VEL
LIN {X 0,Y 51.071,Z 946.918,A -85,B 0,C 180,E1 -29242.079,E2 -29242.079} C_VEL
LIN {X 0,Y 51.481,Z 948.613,A -85,B 0,C 180,E1 -29249.988,E2 -29249.988} C_VEL
LIN {X 0,Y 50.777,Z 949.965,A -85,B 0,C 180,E1 -29264.339,E2 -29264.339} C_VEL
LIN {X 0,Y 51.942,Z 950.19,A -85,B 0,C 180,E1 -29273.936,E2 -29273.936} C_VEL
LIN {X 0,Y 56.907,Z 949.374,A -85,B 0,C 180,E1 -29288.12,E2 -29288.12} C_VEL
LIN {X 0,Y 65.014,Z 947.153,A -85,B 0,C 180,E1 -29299.159,E2 -29299.159} C_VEL
LIN {X 0,Y 75.1,Z 943.456,A -85,B 0,C 180,E1 -29307.362,E2 -29307.362} C_VEL
LIN {X 0,Y 83.543,Z 939.62,A -85,B 0,C 180,E1 -29312.028,E2 -29312.028} C_VEL
LIN {X 0,Y 92.527,Z 934.783,A -85,B 0,C 180,E1 -29315.693,E2 -29315.693} C_VEL
LIN {X 0,Y 103.508,Z 927.689,A -85,B 0,C 180,E1 -29318.985,E2 -29318.985} C_VEL
LIN {X 0,Y 113.186,Z 920.14,A -85,B 0,C 180,E1 -29321.228,E2 -29321.228} C_VEL
LIN {X 0,Y 123.088,Z 910.917,A -85,B 0,C 180,E1 -29322.996,E2 -29322.996} C_VEL
LIN {X 0,Y 132.263,Z 900.469,A -85,B 0,C 180,E1 -29324.368,E2 -29324.368} C_VEL
LIN {X 0,Y 140.712,Z 888.676,A -85,B 0,C 180,E1 -29325.38,E2 -29325.38} C_VEL
LIN {X 0,Y 147.194,Z 877.359,A -85,B 0,C 180,E1 -29326.071,E2 -29326.071} C_VEL
LIN {X 0,Y 152.529,Z 865.493,A -85,B 0,C 180,E1 -29326.571,E2 -29326.571} C_VEL
LIN {X 0,Y 155.463,Z 857.272,A -85,B 0,C 180,E1 -29326.937,E2 -29326.937} C_VEL
LIN {X 0,Y 155.99,Z 854.712,A -85,B 0,C 180,E1 -29329.618,E2 -29329.618} C_VEL
LIN {X 0,Y 156.042,Z 854.753,A -85,B 0,C 180,E1 -29331.257,E2 -29331.257} C_VEL
LIN {X 0,Y 151.458,Z 866.989,A -85,B 0,C 180,E1 -29332.22,E2 -29332.22} C_VEL
LIN {X 0,Y 151.357,Z 867.22,A -85,B 0,C 180,E1 -29332.241,E2 -29332.241} C_VEL
LIN {X 0,Y 148.849,Z 872.625,A -85,B 0,C 180,E1 -29332.48,E2 -29332.48} C_VEL
LIN {X 0,Y 144.083,Z 881.327,A -85,B 0,C 180,E1 -29332.24,E2 -29332.24} C_VEL
LIN {X 0,Y 138.739,Z 889.575,A -85,B 0,C 180,E1 -29332.054,E2 -29332.054} C_VEL
LIN {X 0,Y 135.287,Z 894.206,A -85,B 0,C 180,E1 -29332.413,E2 -29332.413} C_VEL
LIN {X 0,Y 127.184,Z 903.566,A -85,B 0,C 180,E1 -29334.024,E2 -29334.024} C_VEL
LIN {X 0,Y 117.359,Z 912.748,A -85,B 0,C 180,E1 -29336.214,E2 -29336.214} C_VEL
LIN {X 0,Y 107.187,Z 920.417,A -85,B 0,C 180,E1 -29338.865,E2 -29338.865} C_VEL
LIN {X 0,Y 98.418,Z 925.795,A -85,B 0,C 180,E1 -29341.569,E2 -29341.569} C_VEL
LIN {X 0,Y 87.758,Z 931.015,A -85,B 0,C 180,E1 -29345.659,E2 -29345.659} C_VEL
LIN {X 0,Y 78.286,Z 934.563,A -85,B 0,C 180,E1 -29350.344,E2 -29350.344} C_VEL
LIN {X 0,Y 72.426,Z 936.265,A -85,B 0,C 180,E1 -29354.019,E2 -29354.019} C_VEL
LIN {X 0,Y 66.663,Z 937.494,A -85,B 0,C 180,E1 -29358.439,E2 -29358.439} C_VEL
LIN {X 0,Y 61.351,Z 938.263,A -85,B 0,C 180,E1 -29363.615,E2 -29363.615} C_VEL
LIN {X 0,Y 56.413,Z 938.564,A -85,B 0,C 180,E1 -29369.891,E2 -29369.891} C_VEL
LIN {X 0,Y 52.499,Z 938.38,A -85,B 0,C 180,E1 -29376.582,E2 -29376.582} C_VEL
LIN {X 0,Y 48.78,Z 937.602,A -85,B 0,C 180,E1 -29386.087,E2 -29386.087} C_VEL
LIN {X 0,Y 45.89,Z 935.101,A -85,B 0,C 180,E1 -29402.663,E2 -29402.663} C_VEL
LIN {X 0,Y 46.399,Z 931.876,A -85,B 0,C 180,E1 -29416.881,E2 -29416.881} C_VEL
LIN {X 0,Y 49.375,Z 927.522,A -85,B 0,C 180,E1 -29430.012,E2 -29430.012} C_VEL
LIN {X 0,Y 54.368,Z 921.931,A -85,B 0,C 180,E1 -29441.192,E2 -29441.192} C_VEL
LIN {X 0,Y 60.742,Z 914.915,A -85,B 0,C 180,E1 -29450.321,E2 -29450.321} C_VEL
LIN {X 0,Y 68.126,Z 906.224,A -85,B 0,C 180,E1 -29457.67,E2 -29457.67} C_VEL
LIN {X 0,Y 74.942,Z 897.177,A -85,B 0,C 180,E1 -29462.801,E2 -29462.801} C_VEL
LIN {X 0,Y 80.324,Z 889.013,A -85,B 0,C 180,E1 -29466.091,E2 -29466.091} C_VEL
LIN {X 0,Y 79.475,Z 888.814,A -85,B 0,C 180,E1 -29467.261,E2 -29467.261} C_VEL
LIN {X 0,Y 74.005,Z 891.948,A -85,B 0,C 180,E1 -29470.557,E2 -29470.557} C_VEL
LIN {X 0,Y 68.469,Z 895.569,A -85,B 0,C 180,E1 -29474.067,E2 -29474.067} C_VEL
LIN {X 0,Y 55.628,Z 903.482,A -85,B 0,C 180,E1 -29489.644,E2 -29489.644} C_VEL
LIN {X 0,Y 52.984,Z 905.484,A -85,B 0,C 180,E1 -29496.55,E2 -29496.55} C_VEL
LIN {X 0,Y 50.749,Z 907.889,A -85,B 0,C 180,E1 -29503.919,E2 -29503.919} C_VEL
LIN {X 0,Y 51.065,Z 913.337,A -85,B 0,C 180,E1 -29527.909,E2 -29527.909} C_VEL
LIN {X 0,Y 56.212,Z 916.525,A -85,B 0,C 180,E1 -29542.028,E2 -29542.028} C_VEL
LIN {X 0,Y 59.551,Z 917.413,A -85,B 0,C 180,E1 -29546.267,E2 -29546.267} C_VEL
LIN {X 0,Y 67.803,Z 924.575,A -85,B 0,C 180,E1 -29553.965,E2 -29553.965} C_VEL
LIN {X 0,Y 68.554,Z 925.247,A -85,B 0,C 180,E1 -29554.887,E2 -29554.887} C_VEL
LIN {X 0,Y 64.625,Z 924.1,A -85,B 0,C 180,E1 -29558.886,E2 -29558.886} C_VEL
LIN {X 0,Y 55.791,Z 931.523,A -85,B 0,C 180,E1 -29566.131,E2 -29566.131} C_VEL
LIN {X 0,Y 49.573,Z 937.308,A -85,B 0,C 180,E1 -29575.438,E2 -29575.438} C_VEL
LIN {X 0,Y 45.23,Z 942.448,A -85,B 0,C 180,E1 -29588.795,E2 -29588.795} C_VEL
LIN {X 0,Y 44.057,Z 945.54,A -85,B 0,C 180,E1 -29600.807,E2 -29600.807} C_VEL
LIN {X 0,Y 44.399,Z 947.345,A -85,B 0,C 180,E1 -29609.986,E2 -29609.986} C_VEL
LIN {X 0,Y 43.877,Z 948.772,A -85,B 0,C 180,E1 -29626.05,E2 -29626.05} C_VEL
LIN {X 0,Y 45.51,Z 949.073,A -85,B 0,C 180,E1 -29637.584,E2 -29637.584} C_VEL
LIN {X 0,Y 51.473,Z 948.426,A -85,B 0,C 180,E1 -29653.037,E2 -29653.037} C_VEL
LIN {X 0,Y 60.597,Z 946.335,A -85,B 0,C 180,E1 -29664.26,E2 -29664.26} C_VEL
LIN {X 0,Y 71.504,Z 942.796,A -85,B 0,C 180,E1 -29672.183,E2 -29672.183} C_VEL
LIN {X 0,Y 80.449,Z 939.082,A -85,B 0,C 180,E1 -29676.511,E2 -29676.511} C_VEL
LIN {X 0,Y 89.837,Z 934.39,A -85,B 0,C 180,E1 -29679.825,E2 -29679.825} C_VEL
LIN {X 0,Y 101.176,Z 927.537,A -85,B 0,C 180,E1 -29682.747,E2 -29682.747} C_VEL
LIN {X 0,Y 111.108,Z 920.215,A -85,B 0,C 180,E1 -29684.691,E2 -29684.691} C_VEL
LIN {X 0,Y 121.209,Z 911.249,A -85,B 0,C 180,E1 -29686.195,E2 -29686.195} C_VEL
LIN {X 0,Y 130.539,Z 901.202,A -85,B 0,C 180,E1 -29687.351,E2 -29687.351} C_VEL
LIN {X 0,Y 138.245,Z 891.095,A -85,B 0,C 180,E1 -29688.107,E2 -29688.107} C_VEL
LIN {X 0,Y 145.332,Z 879.63,A -85,B 0,C 180,E1 -29688.733,E2 -29688.733} C_VEL
LIN {X 0,Y 151.412,Z 867.19,A -85,B 0,C 180,E1 -29689.187,E2 -29689.187} C_VEL
LIN {X 0,Y 152.107,Z 865.49,A -85,B 0,C 180,E1 -29689.35,E2 -29689.35} C_VEL
LIN {X 0,Y 147.058,Z 876.155,A -85,B 0,C 180,E1 -29690.266,E2 -29690.266} C_VEL
LIN {X 0,Y 140.803,Z 886.586,A -85,B 0,C 180,E1 -29691.389,E2 -29691.389} C_VEL
LIN {X 0,Y 135.287,Z 894.206,A -85,B 0,C 180,E1 -29692.413,E2 -29692.413} C_VEL
LIN {X 0,Y 132.812,Z 897.32,A -85,B 0,C 180,E1 -29692.589,E2 -29692.589} C_VEL
LIN {X 0,Y 128.446,Z 902.386,A -85,B 0,C 180,E1 -29692.128,E2 -29692.128} C_VEL
LIN {X 0,Y 123.854,Z 907.223,A -85,B 0,C 180,E1 -29691.66,E2 -29691.66} C_VEL
LIN {X 0,Y 120.971,Z 909.927,A -85,B 0,C 180,E1 -29691.872,E2 -29691.872} C_VEL
LIN {X 0,Y 111.318,Z 917.786,A -85,B 0,C 180,E1 -29693.863,E2 -29693.863} C_VEL
LIN {X 0,Y 101.154,Z 924.449,A -85,B 0,C 180,E1 -29696.334,E2 -29696.334} C_VEL
LIN {X 0,Y 91.363,Z 929.604,A -85,B 0,C 180,E1 -29699.161,E2 -29699.161} C_VEL
LIN {X 0,Y 80.924,Z 933.893,A -85,B 0,C 180,E1 -29703.036,E2 -29703.036} C_VEL
LIN {X 0,Y 70.939,Z 936.923,A -85,B 0,C 180,E1 -29707.882,E2 -29707.882} C_VEL
LIN {X 0,Y 63.264,Z 938.533,A -85,B 0,C 180,E1 -29712.838,E2 -29712.838} C_VEL
LIN {X 0,Y 53.182,Z 939.581,A -85,B 0,C 180,E1 -29722.354,E2 -29722.354} C_VEL
LIN {X 0,Y 48.295,Z 939.528,A -85,B 0,C 180,E1 -29729.201,E2 -29729.201} C_VEL
LIN {X 0,Y 42.797,Z 938.673,A -85,B 0,C 180,E1 -29741.063,E2 -29741.063} C_VEL
LIN {X 0,Y 39.237,Z 936.581,A -85,B 0,C 180,E1 -29757.515,E2 -29757.515} C_VEL
LIN {X 0,Y 39.015,Z 933.532,A -85,B 0,C 180,E1 -29774.34,E2 -29774.34} C_VEL
LIN {X 0,Y 42.181,Z 928.926,A -85,B 0,C 180,E1 -29791.319,E2 -29791.319} C_VEL
LIN {X 0,Y 48.055,Z 922.966,A -85,B 0,C 180,E1 -29804.842,E2 -29804.842} C_VEL
LIN {X 0,Y 55.055,Z 915.948,A -85,B 0,C 180,E1 -29814.523,E2 -29814.523} C_VEL
LIN {X 0,Y 63.053,Z 907.248,A -85,B 0,C 180,E1 -29821.979,E2 -29821.979} C_VEL
LIN {X 0,Y 70.562,Z 897.881,A -85,B 0,C 180,E1 -29827.172,E2 -29827.172} C_VEL
LIN {X 0,Y 70.709,Z 897.628,A -85,B 0,C 180,E1 -29827.329,E2 -29827.329} C_VEL
LIN {X 0,Y 64.973,Z 900.854,A -85,B 0,C 180,E1 -29830.782,E2 -29830.782} C_VEL
LIN {X 0,Y 51.161,Z 908.332,A -85,B 0,C 180,E1 -29846.667,E2 -29846.667} C_VEL
LIN {X 0,Y 45.616,Z 912.587,A -85,B 0,C 180,E1 -29862.051,E2 -29862.051} C_VEL
LIN {X 0,Y 45.662,Z 917.883,A -85,B 0,C 180,E1 -29888.852,E2 -29888.852} C_VEL
LIN {X 0,Y 51.15,Z 920.969,A -85,B 0,C 180,E1 -29904.342,E2 -29904.342} C_VEL
LIN {X 0,Y 55.439,Z 922.093,A -85,B 0,C 180,E1 -29910.468,E2 -29910.468} C_VEL
LIN {X 0,Y 57.768,Z 923.046,A -85,B 0,C 180,E1 -29913.758,E2 -29913.758} C_VEL
LIN {X 0,Y 58.006,Z 923.975,A -85,B 0,C 180,E1 -29915.334,E2 -29915.334} C_VEL
LIN {X 0,Y 49.73,Z 930.813,A -85,B 0,C 180,E1 -29922.085,E2 -29922.085} C_VEL
LIN {X 0,Y 42.082,Z 937.383,A -85,B 0,C 180,E1 -29934.213,E2 -29934.213} C_VEL
LIN {X 0,Y 38.088,Z 941.791,A -85,B 0,C 180,E1 -29948.327,E2 -29948.327} C_VEL
LIN {X 0,Y 37.079,Z 944.132,A -85,B 0,C 180,E1 -29959.058,E2 -29959.058} C_VEL
LIN {X 0,Y 37.322,Z 946.015,A -85,B 0,C 180,E1 -29969.984,E2 -29969.984} C_VEL
LIN {X 0,Y 37.061,Z 947.543,A -85,B 0,C 180,E1 -29988.533,E2 -29988.533} C_VEL
LIN {X 0,Y 39.307,Z 947.954,A -85,B 0,C 180,E1 -30002.42,E2 -30002.42} C_VEL
LIN {X 0,Y 46.511,Z 947.434,A -85,B 0,C 180,E1 -30019.051,E2 -30019.051} C_VEL
LIN {X 0,Y 56.716,Z 945.526,A -85,B 0,C 180,E1 -30030.138,E2 -30030.138} C_VEL
LIN {X 0,Y 68.458,Z 942.117,A -85,B 0,C 180,E1 -30037.488,E2 -30037.488} C_VEL
LIN {X 0,Y 81.092,Z 937.172,A -85,B 0,C 180,E1 -30042.402,E2 -30042.402} C_VEL
LIN {X 0,Y 90.942,Z 932.305,A -85,B 0,C 180,E1 -30044.99,E2 -30044.99} C_VEL
LIN {X 0,Y 102.665,Z 925.152,A -85,B 0,C 180,E1 -30047.26,E2 -30047.26} C_VEL
LIN {X 0,Y 112.86,Z 917.562,A -85,B 0,C 180,E1 -30048.72,E2 -30048.72} C_VEL
LIN {X 0,Y 123.161,Z 908.283,A -85,B 0,C 180,E1 -30049.818,E2 -30049.818} C_VEL
LIN {X 0,Y 128.316,Z 902.795,A -85,B 0,C 180,E1 -30050.33,E2 -30050.33} C_VEL
LIN {X 0,Y 128.231,Z 902.843,A -85,B 0,C 180,E1 -30050.555,E2 -30050.555} C_VEL
LIN {X 0,Y 120.971,Z 909.927,A -85,B 0,C 180,E1 -30051.872,E2 -30051.872} C_VEL
LIN {X 0,Y 116.12,Z 914.136,A -85,B 0,C 180,E1 -30052.483,E2 -30052.483} C_VEL
LIN {X 0,Y 103.776,Z 923.21,A -85,B 0,C 180,E1 -30052.824,E2 -30052.824} C_VEL
LIN {X 0,Y 96.339,Z 927.639,A -85,B 0,C 180,E1 -30053.378,E2 -30053.378} C_VEL
LIN {X 0,Y 92.641,Z 929.501,A -85,B 0,C 180,E1 -30054.094,E2 -30054.094} C_VEL
LIN {X 0,Y 80.888,Z 934.404,A -85,B 0,C 180,E1 -30057.506,E2 -30057.506} C_VEL
LIN {X 0,Y 70.296,Z 937.599,A -85,B 0,C 180,E1 -30061.587,E2 -30061.587} C_VEL
LIN {X 0,Y 60.58,Z 939.571,A -85,B 0,C 180,E1 -30066.663,E2 -30066.663} C_VEL
LIN {X 0,Y 50.731,Z 940.574,A -85,B 0,C 180,E1 -30074.18,E2 -30074.18} C_VEL
LIN {X 0,Y 45.022,Z 940.632,A -85,B 0,C 180,E1 -30080.548,E2 -30080.548} C_VEL
LIN {X 0,Y 37.307,Z 939.745,A -85,B 0,C 180,E1 -30094.415,E2 -30094.415} C_VEL
LIN {X 0,Y 33.016,Z 938.019,A -85,B 0,C 180,E1 -30110.337,E2 -30110.337} C_VEL
LIN {X 0,Y 31.709,Z 935.152,A -85,B 0,C 180,E1 -30130.602,E2 -30130.602} C_VEL
LIN {X 0,Y 34.201,Z 931.173,A -85,B 0,C 180,E1 -30150.018,E2 -30150.018} C_VEL
LIN {X 0,Y 39.698,Z 925.971,A -85,B 0,C 180,E1 -30165.415,E2 -30165.415} C_VEL
LIN {X 0,Y 47.938,Z 918.631,A -85,B 0,C 180,E1 -30177.673,E2 -30177.673} C_VEL
LIN {X 0,Y 55.44,Z 911.372,A -85,B 0,C 180,E1 -30184.795,E2 -30184.795} C_VEL
LIN {X 0,Y 59.22,Z 907.373,A -85,B 0,C 180,E1 -30187.579,E2 -30187.579} C_VEL
LIN {X 0,Y 58.444,Z 907.181,A -85,B 0,C 180,E1 -30189.382,E2 -30189.382} C_VEL
LIN {X 0,Y 46.659,Z 912.869,A -85,B 0,C 180,E1 -30202.949,E2 -30202.949} C_VEL
LIN {X 0,Y 40.31,Z 916.944,A -85,B 0,C 180,E1 -30219.59,E2 -30219.59} C_VEL
LIN {X 0,Y 40.038,Z 922.098,A -85,B 0,C 180,E1 -30250.108,E2 -30250.108} C_VEL
LIN {X 0,Y 47.603,Z 925.511,A -85,B 0,C 180,E1 -30269.889,E2 -30269.889} C_VEL
LIN {X 0,Y 48.466,Z 925.719,A -85,B 0,C 180,E1 -30271.109,E2 -30271.109} C_VEL
LIN {X 0,Y 47.765,Z 927.175,A -85,B 0,C 180,E1 -30273.48,E2 -30273.48} C_VEL
LIN {X 0,Y 41.36,Z 932.105,A -85,B 0,C 180,E1 -30280.102,E2 -30280.102} C_VEL
LIN {X 0,Y 34.644,Z 937.376,A -85,B 0,C 180,E1 -30292.491,E2 -30292.491} C_VEL
LIN {X 0,Y 30.683,Z 941.558,A -85,B 0,C 180,E1 -30309.885,E2 -30309.885} C_VEL
LIN {X 0,Y 30.244,Z 944.671,A -85,B 0,C 180,E1 -30329.98,E2 -30329.98} C_VEL
LIN {X 0,Y 30.318,Z 946.269,A -85,B 0,C 180,E1 -30351.996,E2 -30351.996} C_VEL
LIN {X 0,Y 33.498,Z 946.832,A -85,B 0,C 180,E1 -30368.983,E2 -30368.983} C_VEL
LIN {X 0,Y 42.179,Z 946.438,A -85,B 0,C 180,E1 -30386.395,E2 -30386.395} C_VEL
LIN {X 0,Y 53.513,Z 944.685,A -85,B 0,C 180,E1 -30396.798,E2 -30396.798} C_VEL
LIN {X 0,Y 66.053,Z 941.455,A -85,B 0,C 180,E1 -30403.221,E2 -30403.221} C_VEL
LIN {X 0,Y 79.229,Z 936.682,A -85,B 0,C 180,E1 -30407.32,E2 -30407.32} C_VEL
LIN {X 0,Y 89.364,Z 931.965,A -85,B 0,C 180,E1 -30409.398,E2 -30409.398} C_VEL
LIN {X 0,Y 99.616,Z 926.139,A -85,B 0,C 180,E1 -30410.968,E2 -30410.968} C_VEL
LIN {X 0,Y 101.533,Z 924.784,A -85,B 0,C 180,E1 -30412.043,E2 -30412.043} C_VEL
LIN {X 0,Y 92.641,Z 929.501,A -85,B 0,C 180,E1 -30414.094,E2 -30414.094} C_VEL
LIN {X 0,Y 87.45,Z 931.943,A -85,B 0,C 180,E1 -30415.027,E2 -30415.027} C_VEL
LIN {X 0,Y 74.502,Z 936.924,A -85,B 0,C 180,E1 -30415.782,E2 -30415.782} C_VEL
LIN {X 0,Y 66.987,Z 939.055,A -85,B 0,C 180,E1 -30416.745,E2 -30416.745} C_VEL
LIN {X 0,Y 63.375,Z 939.824,A -85,B 0,C 180,E1 -30417.888,E2 -30417.888} C_VEL
LIN {X 0,Y 56.226,Z 940.949,A -85,B 0,C 180,E1 -30421.22,E2 -30421.22} C_VEL
LIN {X 0,Y 44.85,Z 941.73,A -85,B 0,C 180,E1 -30429.017,E2 -30429.017} C_VEL
LIN {X 0,Y 36.914,Z 941.411,A -85,B 0,C 180,E1 -30437.892,E2 -30437.892} C_VEL
LIN {X 0,Y 31.654,Z 940.643,A -85,B 0,C 180,E1 -30447.407,E2 -30447.407} C_VEL
LIN {X 0,Y 27.513,Z 939.412,A -85,B 0,C 180,E1 -30460.01,E2 -30460.01} C_VEL
LIN {X 0,Y 24.93,Z 937.542,A -85,B 0,C 180,E1 -30477.757,E2 -30477.757} C_VEL
LIN {X 0,Y 25.42,Z 934.319,A -85,B 0,C 180,E1 -30502.078,E2 -30502.078} C_VEL
LIN {X 0,Y 30.193,Z 929.731,A -85,B 0,C 180,E1 -30523.481,E2 -30523.481} C_VEL
LIN {X 0,Y 37.667,Z 923.863,A -85,B 0,C 180,E1 -30537.822,E2 -30537.822} C_VEL
LIN {X 0,Y 46.438,Z 916.577,A -85,B 0,C 180,E1 -30547.271,E2 -30547.271} C_VEL
LIN {X 0,Y 47.865,Z 915.333,A -85,B 0,C 180,E1 -30548.422,E2 -30548.422} C_VEL
LIN {X 0,Y 47.943,Z 914.601,A -85,B 0,C 180,E1 -30550.748,E2 -30550.748} C_VEL
LIN {X 0,Y 34.876,Z 920.982,A -85,B 0,C 180,E1 -30576.23,E2 -30576.23} C_VEL
LIN {X 0,Y 34.201,Z 925.945,A -85,B 0,C 180,E1 -30611.856,E2 -30611.856} C_VEL
LIN {X 0,Y 39.112,Z 928.258,A -85,B 0,C 180,E1 -30627.775,E2 -30627.775} C_VEL
LIN {X 0,Y 38.473,Z 929.514,A -85,B 0,C 180,E1 -30630.599,E2 -30630.599} C_VEL
LIN {X 0,Y 29.381,Z 935.76,A -85,B 0,C 180,E1 -30644.115,E2 -30644.115} C_VEL
LIN {X 0,Y 24.171,Z 940.071,A -85,B 0,C 180,E1 -30664.114,E2 -30664.114} C_VEL
LIN {X 0,Y 23.162,Z 943.312,A -85,B 0,C 180,E1 -30689.974,E2 -30689.974} C_VEL
LIN {X 0,Y 23.745,Z 944.983,A -85,B 0,C 180,E1 -30717.392,E2 -30717.392} C_VEL
LIN {X 0,Y 28.317,Z 945.686,A -85,B 0,C 180,E1 -30738.091,E2 -30738.091} C_VEL
LIN {X 0,Y 38.689,Z 945.443,A -85,B 0,C 180,E1 -30755.228,E2 -30755.228} C_VEL
LIN {X 0,Y 51.128,Z 943.828,A -85,B 0,C 180,E1 -30764.153,E2 -30764.153} C_VEL
LIN {X 0,Y 64.358,Z 940.799,A -85,B 0,C 180,E1 -30769.308,E2 -30769.308} C_VEL
LIN {X 0,Y 77.976,Z 936.179,A -85,B 0,C 180,E1 -30772.435,E2 -30772.435} C_VEL
LIN {X 0,Y 77.876,Z 936.126,A -85,B 0,C 180,E1 -30773.006,E2 -30773.006} C_VEL
LIN {X 0,Y 70.514,Z 938.275,A -85,B 0,C 180,E1 -30775.221,E2 -30775.221} C_VEL
LIN {X 0,Y 63.375,Z 939.824,A -85,B 0,C 180,E1 -30777.888,E2 -30777.888} C_VEL
LIN {X 0,Y 57.878,Z 940.896,A -85,B 0,C 180,E1 -30779.684,E2 -30779.684} C_VEL
LIN {X 0,Y 48.184,Z 942.178,A -85,B 0,C 180,E1 -30781.533,E2 -30781.533} C_VEL
LIN {X 0,Y 40.366,Z 942.603,A -85,B 0,C 180,E1 -30783.403,E2 -30783.403} C_VEL
LIN {X 0,Y 34.8,Z 942.515,A -85,B 0,C 180,E1 -30786.5,E2 -30786.5} C_VEL
LIN {X 0,Y 33.091,Z 942.343,A -85,B 0,C 180,E1 -30788.152,E2 -30788.152} C_VEL
LIN {X 0,Y 28.613,Z 941.87,A -85,B 0,C 180,E1 -30794.221,E2 -30794.221} C_VEL
LIN {X 0,Y 23.327,Z 940.787,A -85,B 0,C 180,E1 -30805.393,E2 -30805.393} C_VEL
LIN {X 0,Y 18.332,Z 938.609,A -85,B 0,C 180,E1 -30830.067,E2 -30830.067} C_VEL
LIN {X 0,Y 18.993,Z 934.598,A -85,B 0,C 180,E1 -30870.032,E2 -30870.032} C_VEL
LIN {X 0,Y 25.446,Z 929.799,A -85,B 0,C 180,E1 -30894.5,E2 -30894.5} C_VEL
LIN {X 0,Y 34.319,Z 923.722,A -85,B 0,C 180,E1 -30907.927,E2 -30907.927} C_VEL
LIN {X 0,Y 36.981,Z 921.771,A -85,B 0,C 180,E1 -30910.517,E2 -30910.517} C_VEL
LIN {X 0,Y 37.932,Z 920.918,A -85,B 0,C 180,E1 -30912.171,E2 -30912.171} C_VEL
LIN {X 0,Y 29.432,Z 924.676,A -85,B 0,C 180,E1 -30931.471,E2 -30931.471} C_VEL
LIN {X 0,Y 29.492,Z 930.097,A -85,B 0,C 180,E1 -30980.321,E2 -30980.321} C_VEL
LIN {X 0,Y 29.48,Z 931.441,A -85,B 0,C 180,E1 -30986.167,E2 -30986.167} C_VEL
LIN {X 0,Y 20.011,Z 937.187,A -85,B 0,C 180,E1 -31005.336,E2 -31005.336} C_VEL
LIN {X 0,Y 16.012,Z 940.915,A -85,B 0,C 180,E1 -31037.285,E2 -31037.285} C_VEL
LIN {X 0,Y 16.084,Z 941.943,A -85,B 0,C 180,E1 -31049.963,E2 -31049.963} C_VEL
LIN {X 0,Y 17.542,Z 943.664,A -85,B 0,C 180,E1 -31086.753,E2 -31086.753} C_VEL
LIN {X 0,Y 24.153,Z 944.501,A -85,B 0,C 180,E1 -31110.751,E2 -31110.751} C_VEL
LIN {X 0,Y 36.284,Z 944.441,A -85,B 0,C 180,E1 -31125.505,E2 -31125.505} C_VEL
LIN {X 0,Y 49.655,Z 942.97,A -85,B 0,C 180,E1 -31132.108,E2 -31132.108} C_VEL
LIN {X 0,Y 53.149,Z 942.214,A -85,B 0,C 180,E1 -31134.633,E2 -31134.633} C_VEL
LIN {X 0,Y 42.158,Z 942.78,A -85,B 0,C 180,E1 -31140.389,E2 -31140.389} C_VEL
LIN {X 0,Y 33.091,Z 942.343,A -85,B 0,C 180,E1 -31148.152,E2 -31148.152} C_VEL
LIN {X 0,Y 27.932,Z 941.921,A -85,B 0,C 180,E1 -31153.502,E2 -31153.502} C_VEL
LIN {X 0,Y 19.03,Z 940.722,A -85,B 0,C 180,E1 -31164.026,E2 -31164.026} C_VEL
LIN {X 0,Y 12.815,Z 939.246,A -85,B 0,C 180,E1 -31181.548,E2 -31181.548} C_VEL
LIN {X 0,Y 10.544,Z 937.708,A -85,B 0,C 180,E1 -31207.68,E2 -31207.68} C_VEL
LIN {X 0,Y 10.646,Z 937.094,A -85,B 0,C 180,E1 -31217.863,E2 -31217.863} C_VEL
LIN {X 0,Y 15.836,Z 933.317,A -85,B 0,C 180,E1 -31256.389,E2 -31256.389} C_VEL
LIN {X 0,Y 26.204,Z 927.356,A -85,B 0,C 180,E1 -31274.842,E2 -31274.842} C_VEL
LIN {X 0,Y 25.253,Z 927.516,A -85,B 0,C 180,E1 -31280.665,E2 -31280.665} C_VEL
LIN {X 0,Y 21.465,Z 932.23,A -85,B 0,C 180,E1 -31333.882,E2 -31333.882} C_VEL
LIN {X 0,Y 18.842,Z 934.071,A -85,B 0,C 180,E1 -31341.113,E2 -31341.113} C_VEL
LIN {X 0,Y 10.727,Z 938.295,A -85,B 0,C 180,E1 -31368.992,E2 -31368.992} C_VEL
LIN {X 0,Y 9.025,Z 940.524,A -85,B 0,C 180,E1 -31409.933,E2 -31409.933} C_VEL
LIN {X 0,Y 12.381,Z 942.304,A -85,B 0,C 180,E1 -31465.421,E2 -31465.421} C_VEL
LIN {X 0,Y 21.587,Z 943.31,A -85,B 0,C 180,E1 -31487.475,E2 -31487.475} C_VEL
LIN {X 0,Y 28.29,Z 943.514,A -85,B 0,C 180,E1 -31493.38,E2 -31493.38} C_VEL
LIN {X 0,Y 30.726,Z 943.42,A -85,B 0,C 180,E1 -31496.131,E2 -31496.131} C_VEL
LIN {X 0,Y 21.197,Z 942.143,A -85,B 0,C 180,E1 -31506.199,E2 -31506.199} C_VEL
LIN {X 0,Y 12.473,Z 939.689,A -85,B 0,C 180,E1 -31534.302,E2 -31534.302} C_VEL
LIN {X 0,Y 10.646,Z 937.094,A -85,B 0,C 180,E1 -31577.863,E2 -31577.863} C_VEL
LIN {X 0,Y 10.717,Z 936.333,A -85,B 0,C 180,E1 -31591.721,E2 -31591.721} C_VEL
LIN {X 0,Y 12.129,Z 934.027,A -85,B 0,C 180,E1 -31637.97,E2 -31637.97} C_VEL
LIN {X 0,Y 14.21,Z 933.004,A -85,B 0,C 180,E1 -31644.012,E2 -31644.012} C_VEL
LIN {X 0,Y 15.479,Z 932.396,A -85,B 0,C 180,E1 -31645.217,E2 -31645.217} C_VEL
LIN {X 0,Y 15.307,Z 932.453,A -85,B 0,C 180,E1 -31652.663,E2 -31652.663} C_VEL
LIN {X 0,Y 13.958,Z 933.98,A -85,B 0,C 180,E1 -31679.995,E2 -31679.995} C_VEL
LIN {X 0,Y 3.824,Z 937.98,A -85,B 0,C 180,E1 -31702.816,E2 -31702.816} C_VEL
LIN {X 0,Y 1.981,Z 939.069,A -85,B 0,C 180,E1 -31769.697,E2 -31769.697} C_VEL
LIN {X 0,Y 7.045,Z 940.484,A -85,B 0,C 180,E1 -31854.892,E2 -31854.892} C_VEL
LIN {X 0,Y 8.775,Z 940.74,A -85,B 0,C 180,E1 -31860.008,E2 -31860.008} C_VEL
LIN {X 0,Y 6.237,Z 936.542,A -85,B 0,C 180,E1 -31984.41,E2 -31984.41} C_VEL
LIN {X 0,Y 14.21,Z 933.004,A -85,B 0,C 180,E1 -32004.012,E2 -32004.012} C_VEL
LIN {X 0,Y 14.21,Z 933.004,A -85,B 0,C 180,E1 -32004.012,E2 -32004.012}

QRS_NEXT_CUT()

QRS_NEXT()
QRS_HOME()

END
